// TIA Portal project "S7_1511_Gantry_Modbus_TCP" (V18)

(* hardware
DEVICE "S7-1500/ET200MP station_1"  S7-1500 station
   slot 0: "Rail_0"  Rack  6ES7 590-1***0-0AA0
   slot 1: "PLC_1"  CPU 1511-1 PN  6ES7 511-1AL03-0AB0  V3.0
      slot 3: "CPU display_1"  6ES7591-1AA00-0AA0
      slot 32768: "PROFINET interface_1"  X1
         slot 32769: "Port_1"  X1 P1
         slot 32770: "Port_2"  X1 P2
      slot 34817: "Virtual CP interface port_1"  Virtual CP interface port  Virtual CP interface port
*)

// ===== PLC "PLC_1"  CPU 1511-1 PN =====

VAR_GLOBAL   // PLC tag table "Default tag table"
   "Clock_Byte" AT %MB0 : Byte;
   "Clock_10Hz" AT %M0.0 : Bool;
   "Clock_5Hz" AT %M0.1 : Bool;
   "Clock_2.5Hz" AT %M0.2 : Bool;
   "Clock_2Hz" AT %M0.3 : Bool;
   "Clock_1.25Hz" AT %M0.4 : Bool;
   "Clock_1Hz" AT %M0.5 : Bool;
   "Clock_0.625Hz" AT %M0.6 : Bool;
   "Clock_0.5Hz" AT %M0.7 : Bool;
   "System_Byte" AT %MB1 : Byte;
   "FirstScan" AT %M1.0 : Bool;
   "DiagStatusUpdate" AT %M1.1 : Bool;
   "AlwaysTRUE" AT %M1.2 : Bool;
   "AlwaysFALSE" AT %M1.3 : Bool;
END_VAR

DATA_BLOCK "DB_Gantry"   // DB2
{ S7_Optimized_Access := 'TRUE' }
VERSION : 0.1
   VAR
      bInXplus : Bool;
      bInXminus : Bool;
      bInYplus : Bool;
      bInYminus : Bool;
      bOutXplus : Bool;
      bOutXminus : Bool;
      bOutYplus : Bool;
      bOutYminus : Bool;
      bEnableXboxController : Bool;
   END_VAR
BEGIN
END_DATA_BLOCK

DATA_BLOCK "DB_ModbusTcpConnect"   // DB10
{ S7_Optimized_Access := 'TRUE' }
VERSION : 0.1
   VAR
      MBTCPClientRead : TCON_IP_v4;
      MBTCPClientRead_DISCONNECT : Bool;
      MBTCPClientRead_DONE : Bool;
      MBTCPClientRead_BUSY : Bool;
      MBTCPClientRead_ERROR : Bool;
      MBTCPClientRead_STATUS : Word;
      MBTCPClientWrite : TCON_IP_v4;
      MBTCPClientWrite_DISCONNECT : Bool;
      MBTCPClientWrite_DONE : Bool;
      MBTCPClientWrite_BUSY : Bool;
      MBTCPClientWrite_ERROR : Bool;
      MBTCPClientWrite_STATUS : Word;
   END_VAR
BEGIN
   MBTCPClientRead.InterfaceId := 64;
   MBTCPClientRead.ID := 16#1;
   MBTCPClientRead.ConnectionType := 16#0B;
   MBTCPClientRead.ActiveEstablished := 1;
   MBTCPClientRead.RemotePort := 502;
   MBTCPClientRead.RemoteAddress.ADDR[1] := 16#C0;
   MBTCPClientRead.RemoteAddress.ADDR[2] := 16#A8;
   MBTCPClientRead.RemoteAddress.ADDR[3] := 16#1;
   MBTCPClientRead.RemoteAddress.ADDR[4] := 16#1F;
   MBTCPClientWrite.InterfaceId := 64;
   MBTCPClientWrite.ID := 16#2;
   MBTCPClientWrite.ConnectionType := 16#0B;
   MBTCPClientWrite.ActiveEstablished := 1;
   MBTCPClientWrite.RemoteAddress.ADDR[1] := 16#C0;
   MBTCPClientWrite.RemoteAddress.ADDR[2] := 16#A8;
   MBTCPClientWrite.RemoteAddress.ADDR[3] := 16#1;
   MBTCPClientWrite.RemoteAddress.ADDR[4] := 16#1F;
   MBTCPClientWrite.RemotePort := 502;
END_DATA_BLOCK

DATA_BLOCK "DB_ModbusTcpData"   // DB11
{ S7_Optimized_Access := 'FALSE' }
VERSION : 0.1
   VAR
      Read : Array[0..19] of Word;
      Write : Array[0..19] of Word;
   END_VAR
BEGIN
END_DATA_BLOCK

FUNCTION "FC_MB_TCP" : Void   // FC10, LAD
{ S7_Optimized_Access := 'TRUE' }
VERSION : 0.1
BEGIN

REGION Network 1
   // Hilfe mit F1 auf Baustein
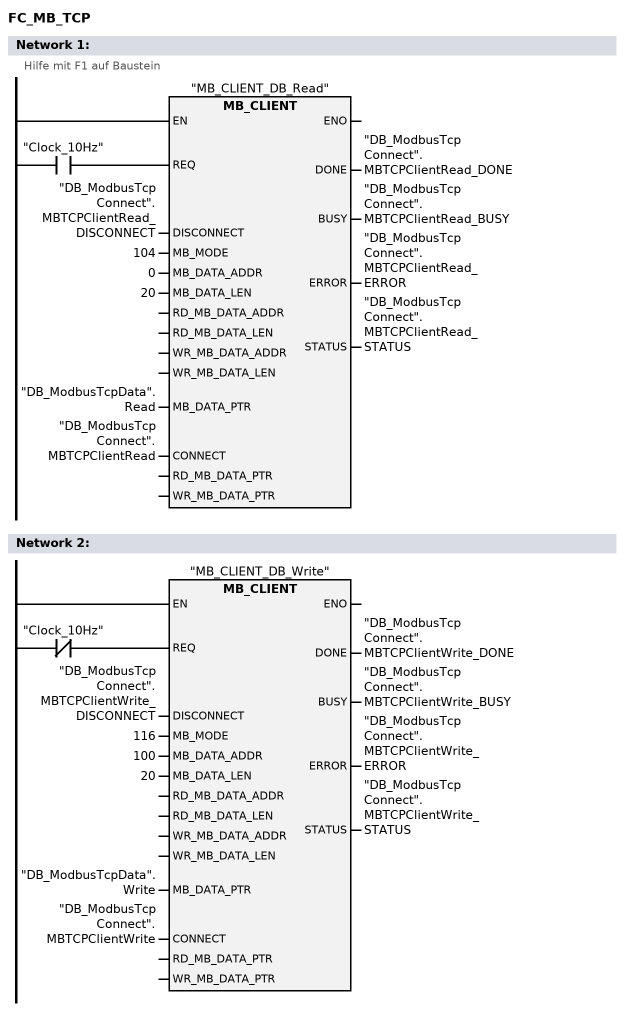
   "MB_CLIENT_DB_Read"(REQ := "Clock_10Hz",   // MB_CLIENT
                       DISCONNECT := "DB_ModbusTcpConnect".MBTCPClientRead_DISCONNECT,
                       MB_MODE := 104,
                       MB_DATA_ADDR := 0,
                       MB_DATA_LEN := 20,
                       MB_DATA_PTR := "DB_ModbusTcpData".Read,
                       CONNECT := "DB_ModbusTcpConnect".MBTCPClientRead,
                       DONE => "DB_ModbusTcpConnect".MBTCPClientRead_DONE,
                       BUSY => "DB_ModbusTcpConnect".MBTCPClientRead_BUSY,
                       ERROR => "DB_ModbusTcpConnect".MBTCPClientRead_ERROR,
                       STATUS => "DB_ModbusTcpConnect".MBTCPClientRead_STATUS);
END_REGION

REGION Network 2
   "MB_CLIENT_DB_Write"(REQ := NOT "Clock_10Hz",   // MB_CLIENT
                        DISCONNECT := "DB_ModbusTcpConnect".MBTCPClientWrite_DISCONNECT,
                        MB_MODE := 116,
                        MB_DATA_ADDR := 100,
                        MB_DATA_LEN := 20,
                        MB_DATA_PTR := "DB_ModbusTcpData".Write,
                        CONNECT := "DB_ModbusTcpConnect".MBTCPClientWrite,
                        DONE => "DB_ModbusTcpConnect".MBTCPClientWrite_DONE,
                        BUSY => "DB_ModbusTcpConnect".MBTCPClientWrite_BUSY,
                        ERROR => "DB_ModbusTcpConnect".MBTCPClientWrite_ERROR,
                        STATUS => "DB_ModbusTcpConnect".MBTCPClientWrite_STATUS);
END_REGION
END_FUNCTION

ORGANIZATION_BLOCK "Main"   // OB1, FBD, ProgramCycle
TITLE = "Main Program Sweep (Cycle)"
{ S7_Optimized_Access := 'TRUE' }
VERSION : 0.1
   VAR_INPUT
      Initial_Call : Bool;   // Initial call of this OB
      Remanence : Bool;   // =True, if remanent data are available
   END_VAR
BEGIN

REGION Network 1
   // Modbusintegration
   // Tutorial ModbusTCP Client via Siemens S7-1200/S7-1500 PLC and TIA Portal: 
   // ttps://www.youtube.com/watch?v=NwzBaDsGpic
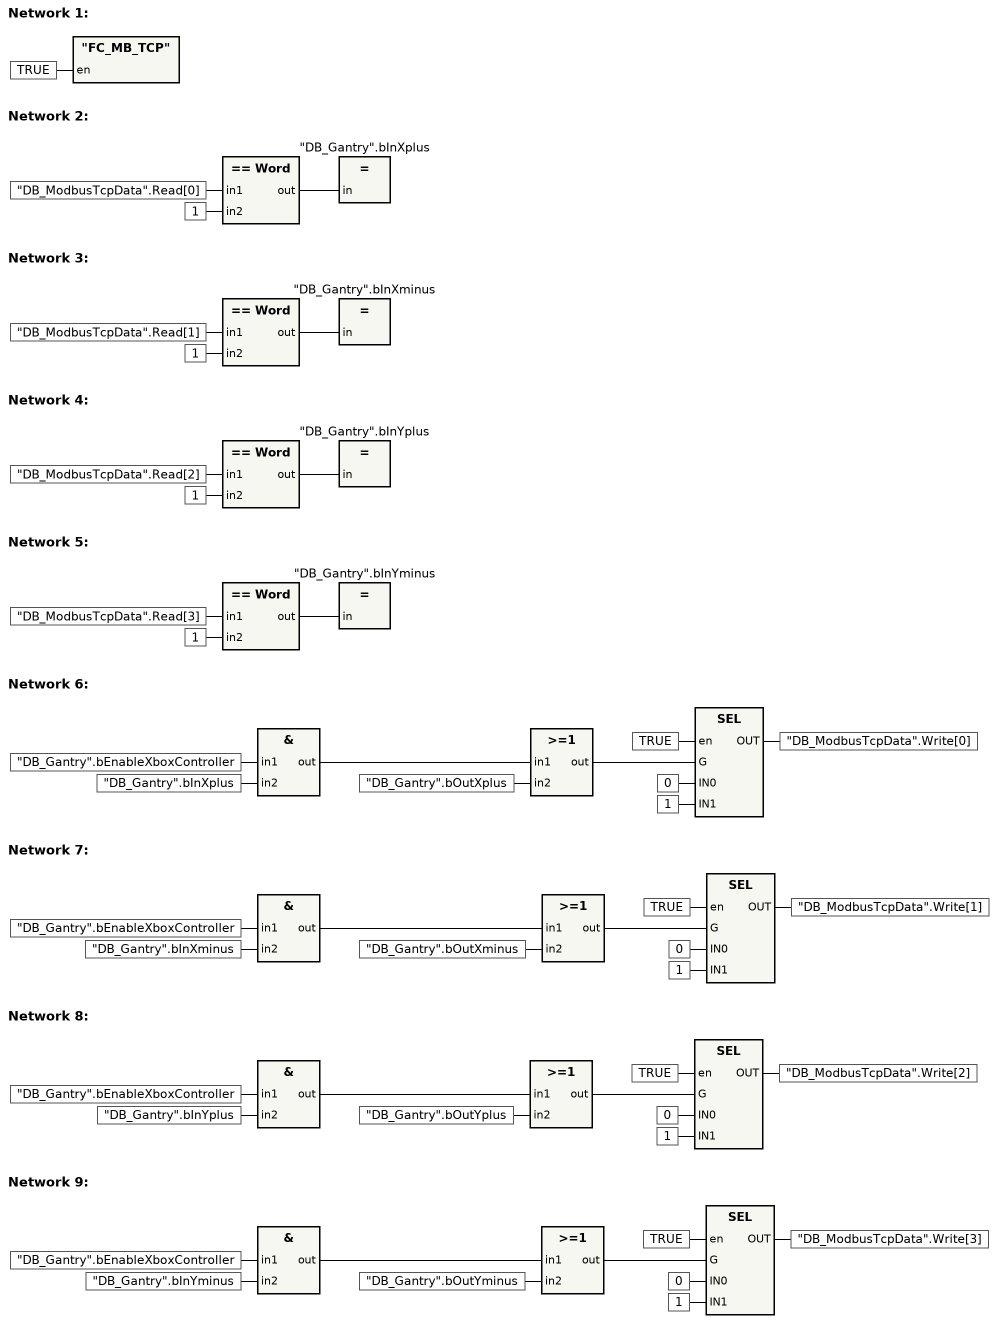
   IF TRUE THEN "FC_MB_TCP"(); END_IF;
END_REGION

REGION Network 2
   "DB_Gantry".bInXplus := "DB_ModbusTcpData".Read[0] = 1;
END_REGION

REGION Network 3
   "DB_Gantry".bInXminus := "DB_ModbusTcpData".Read[1] = 1;
END_REGION

REGION Network 4
   "DB_Gantry".bInYplus := "DB_ModbusTcpData".Read[2] = 1;
END_REGION

REGION Network 5
   "DB_Gantry".bInYminus := "DB_ModbusTcpData".Read[3] = 1;
END_REGION

REGION Network 6
   // X PLUS
   IF TRUE THEN
       "DB_ModbusTcpData".Write[0] := SEL(G := ("DB_Gantry".bEnableXboxController AND "DB_Gantry".bInXplus) OR "DB_Gantry".bOutXplus, IN0 := 0, IN1 := 1);
   END_IF;
END_REGION

REGION Network 7
   // X MINUS
   IF TRUE THEN
       "DB_ModbusTcpData".Write[1] := SEL(G := ("DB_Gantry".bEnableXboxController AND "DB_Gantry".bInXminus) OR "DB_Gantry".bOutXminus, IN0 := 0, IN1 := 1);
   END_IF;
END_REGION

REGION Network 8
   // Y PLUS
   IF TRUE THEN
       "DB_ModbusTcpData".Write[2] := SEL(G := ("DB_Gantry".bEnableXboxController AND "DB_Gantry".bInYplus) OR "DB_Gantry".bOutYplus, IN0 := 0, IN1 := 1);
   END_IF;
END_REGION

REGION Network 9
   // Y MINUS
   IF TRUE THEN
       "DB_ModbusTcpData".Write[3] := SEL(G := ("DB_Gantry".bEnableXboxController AND "DB_Gantry".bInYminus) OR "DB_Gantry".bOutYminus, IN0 := 0, IN1 := 1);
   END_IF;
END_REGION
END_ORGANIZATION_BLOCK